TYPE ST_Circle :
STRUCT
	rX : REAL;
	rY : REAL;
	rD : REAL;
END_STRUCT
END_TYPE

(* stored: Version 1.1.0.1, ProductVersion 3.1.4020.12
   DUT ST_Circle: Id {e6ffb2c9-1b1a-4d6d-b40a-ebea44c15402} *)
